INTERFACE I_XtsTransport_Station

METHOD Init : e_progress
VAR_INPUT
END_VAR
END_METHOD

PROPERTY MessageLevel : e_messagetype
SET
END_SET
END_PROPERTY

PROPERTY StationId : uint // know thy reflection,
GET
END_GET
SET
END_SET
END_PROPERTY

PROPERTY TargetWindow : lreal
GET
END_GET
SET
END_SET
END_PROPERTY

END_INTERFACE

(* stored: Version 1.1.0.1, ProductVersion 3.1.4024.15
   Itf I_XtsTransport_Station: Id {11da36ff-f863-4c10-9d89-4614b0ee2b8d}
   Folder methods: Id {115de0eb-c9ab-4032-ab3a-abe5b5a3f88b}
   Folder properties: Id {657be21a-1910-4d0d-bba7-3dd552a5d261}
   Method Init: Id {07fb410f-6e62-44ba-a6fd-a903ddf1ca81}
   Property MessageLevel: Id {7e6e258b-b152-4962-a065-c206eba09533}
   Set Set: Id {e9994b99-055f-4152-86bf-3d6a569f2bb1}
   Property StationId: Id {7741cf4a-9932-469b-9500-917e4fbfb92d}
   Get Get: Id {6a47f0e9-e898-441c-ac29-b9348bc7feca}
   Set Set: Id {23e8277c-f4fd-45a2-aa62-afa4ec5fb55e}
   Property TargetWindow: Id {28a03c52-644f-49e7-be48-988817d2b05a}
   Get Get: Id {feaad07d-a692-4f5b-b6a2-fcae920f2beb}
   Set Set: Id {4b2d6bcc-3a78-411a-aa37-ef3a36839038} *)
